TYPE st_Robot_Input :
STRUCT
    fault : BOOL;
END_STRUCT
END_TYPE

(* stored: Version 1.1.0.1, ProductVersion 3.1.4024.9
   DUT st_Robot_Input: Id {ce91bbf5-201a-40e8-9f5c-1b913e0b33ac} *)
